(* IEC 61131-3 sources: AXOpen/src/core/ctrl/src/AxoMessaging/Logger, 1 file *)

(* ---- AxoLogger.st ---- *)
USING AXOpen.Core;
USING AXOpen.Messaging;

NAMESPACE AXOpen.Messaging
    CLASS PUBLIC LogEntry
        VAR PUBLIC
            Message : STRING[80];
            Level : eLogLevel;
            Sender : ULINT;
            ToDequeue : BOOL;
        END_VAR
    END_CLASS

    CLASS PUBLIC AxoLogger IMPLEMENTS IAxoLogger, IAxoLoggerConfig
        VAR PUBLIC
            Carret : INT := 0;
            MinLevel : eLogLevel;
            LogEntries : ARRAY[0..100] OF LogEntry;
        END_VAR

        METHOD PUBLIC Log
            VAR_INPUT
                _message : STRING[80];
                _level : eLogLevel;
                _sender : IAxoObject;
            END_VAR

            IF(_level >= THIS.MinLevel) THEN
                IF(Carret > 100) THEN
                    Carret := 0;
                END_IF;

                LogEntries[Carret].Message := _message;
                LogEntries[Carret].Level := _level;

                IF(_sender <> NULL) THEN
                    LogEntries[Carret].Sender := _sender.GetIdentity();
                END_IF;

                LogEntries[Carret].ToDequeue := TRUE;
                Carret := Carret + 1;
            END_IF;
        END_METHOD

        METHOD PUBLIC MinimumLevel : IAxoLoggerConfig
            VAR_INPUT
                _level : eLogLevel;
            END_VAR
            THIS.MinLevel := _level;
            MinimumLevel := THIS;
        END_METHOD
    END_CLASS
END_NAMESPACE
